INTERFACE I_CollectionNode EXTENDS I_Disposable

PROPERTY PUBLIC DataSize : UDINT
GET
END_GET
END_PROPERTY

METHOD PUBLIC Equals : BOOL
VAR_INPUT
	Symbol : ANY;
END_VAR
END_METHOD

METHOD PUBLIC TryGet : BOOL;
VAR_INPUT
	Destination : ANY;
END_VAR
END_METHOD

METHOD PUBLIC TryGetTo : BOOL;
VAR_INPUT
	DestinationAddress : PVOID;
	DestinationSize : UDINT;
END_VAR
END_METHOD

END_INTERFACE

(* stored: Version 1.1.0.1, ProductVersion 3.1.4024.12
   Itf I_CollectionNode: Id {cc06b10f-e542-0eb2-371b-5881da920510}
   Property DataSize: Id {8fb392fd-758c-0751-264a-ed59d6358b2d}
   Get Get: Id {58a11401-376a-004d-1516-8d50469ebdcd}
   Method Equals: Id {3409ed2a-b83d-09b9-0b6f-192cb6a542b6}
   Method TryGet: Id {74e09bfd-a3ab-04a8-3616-8d1e86304b2e}
   Method TryGetTo: Id {248caae0-1b9c-05ce-110c-5e946c6c5d0b} *)
